TYPE Handshake_Receive :
STRUCT
	ReadyToReceive 	: BOOL;
	Received		: BOOL;
	PartInfo		: STRING(20);
END_STRUCT
END_TYPE

(* stored: Version 1.1.0.1, ProductVersion 3.1.4022.11
   DUT Handshake_Receive: Id {da99d67a-2c73-46e1-8180-e4aa491c9fc3} *)
